{attribute 'GeneratedUsingTerminal: EK1122-0000-0018'}
{attribute addProperty BoxType "EK1122-0000-0018"}
{attribute addProperty Id "Beckhoff_EK12xxsub_EK1100EK1100_1FC0878B2"}
{attribute addProperty CRC "4030482601"}
{attribute addProperty Size "2"}
TYPE Beckhoff_EK12xxEK1122_F03C48A9 EXTENDS EK1122_1FC0878B :
STRUCT
	{attribute addProperty Name "Beckhoff EK12xxsub EK1100"}
	{attribute addProperty PreviousPort "Beckhoff EK12xxEK1122 : D"}
	Beckhoff_EK12xxsub_EK1100 : EK1100_1FC0878B;
END_STRUCT
END_TYPE

(* stored: Version 1.2.0.0, ProductVersion 3.1.4024.9
   DUT Beckhoff_EK12xxEK1122_F03C48A9: Id {7ba5ae41-c1ce-4f48-94ef-6710168c1b25} *)
